TYPE Iv3Id01Status :
STRUCT
bit0 : BIT;

END_STRUCT
END_TYPE

(* stored: Version 1.1.0.1, ProductVersion 3.1.4024.12
   DUT Iv3Id01Status: Id {65eb9b97-5cc9-07b2-3d26-40b3590db82b} *)
